// TwinCAT 3 PLC project Core
// Title: MTP
// Company: Zerlauth
// Author: Peter Zerlauth
// ProjectVersion: 0.0.0.0
// Description: Module Type Package MTP
// ProgramVersion: 3.1.4024.0
// libraries:
//   Tc2_Standard, * (Beckhoff Automation GmbH)
//   Tc2_System, * (Beckhoff Automation GmbH)
//   Tc2_Utilities, * (Beckhoff Automation GmbH)
// project tree:
//   Component/Event/ E_Event.TcDUT (not stored), E_Behaviour.TcDUT, FB_Event.TcPOU, I_Event.TcIO, ST_Event.TcDUT
//   Component/ E_Request.TcDUT (not stored), E_State.TcDUT, FB_Component.TcPOU, I_Component.TcIO
//   Component/Info/ FB_Info.TcPOU, I_Info.TcIO
//   Component/Observer/ FB_Observer.TcPOU, I_Observer.TcIO (not stored)
//   CyclicCall/ FB_Cycle.TcPOU, I_Cycle.TcIO
//   List/ FB_ListComponent.TcPOU (not stored), FB_ListObject.TcPOU, FB_ListString.TcPOU (not stored), I_ListComponent.TcIO (not stored), I_ListObject.TcIO, I_ListString.TcIO (not stored)
//   Logger/ FB_ListLogger.TcPOU, I_Logger.TcIO (not stored)
//   Object/ I_Object.TcIO (not stored)
//   Sequence/ FB_Sequence.TcPOU (not stored), I_Sequence.TcIO (not stored)
// (motion and I/O tree: see PLC project example)
// real-time tasks:
//   TASK plcTask1: cycle T#25000us, priority 20, ADS port 350

// ---- Component/Event/E_Behaviour.TcDUT
{attribute 'qualified_only'}
{attribute 'strict'}
{attribute 'to_string'}
TYPE E_Behaviour :
(
    Pause    := 100,
    Hold     := 200,    
	Complete := 300,	
    Stop  	 := 400,    
	Abort    := 500
 );	
END_TYPE

// ---- Component/Event/ST_Event.TcDUT
TYPE ST_Event :
STRUCT
	Source:			I_Component;
	EventType:		E_Event;
	Timestamp:   	ULINT;
	ID:				UDINT;
	Message:		STRING(255);
	Arguments:		STRING(255);
	Active:		BOOL;
END_STRUCT
END_TYPE

// ---- Component/E_State.TcDUT
{attribute 'qualified_only'}
{attribute 'strict'}
{attribute 'to_string'}
TYPE E_State :
(
	{attribute 'hide'}
	Undefined		:= 0,
	Idle			:= 1,
	
// Start
	Starting		:= 2,
	Execute			:= 3,
	
// Pause
	Pausing			:= 4,
	Paused			:= 5,
	Resuming		:= 6,
	
// Hold
	Holding			:= 7,
	Held			:= 8,
	Unholding		:= 9,
	
// Complete
	Completing		:= 10,
	Completed		:= 11,

// Stop
	Stopping		:= 12,
	Stopped			:= 13,

// Abort	
	Aborting		:= 14,
	Aborted			:= 15,

// Reset
	Resetting		:= 16

);
END_TYPE

// ---- Component/Event/I_Event.TcIO
INTERFACE I_Event EXTENDS I_Object

METHOD PUBLIC M_Debug : BOOL
VAR_INPUT
	Message:				STRING(255);
END_VAR
END_METHOD

METHOD PUBLIC M_Error : BOOL
VAR_INPUT
	Message:				STRING(255);
	ID:						UDINT;
	Behaviour:				E_Behaviour;
END_VAR
END_METHOD

METHOD PUBLIC M_Information : BOOL
VAR_INPUT
	Message:				STRING(255);
	ID:						UDINT;
END_VAR
END_METHOD

METHOD PUBLIC M_Warning : BOOL
VAR_INPUT
	Message:				STRING(255);
	ID:						UDINT;
END_VAR
END_METHOD

PROPERTY PUBLIC P_Logger : I_Logger
GET
END_GET
SET
END_SET
END_PROPERTY

END_INTERFACE

// ---- Component/Info/I_Info.TcIO
INTERFACE I_Info EXTENDS I_Object

PROPERTY PUBLIC P_Class : String(255)
GET
END_GET
END_PROPERTY

PROPERTY PUBLIC P_Comment : String(255)
GET
END_GET
END_PROPERTY

PROPERTY PUBLIC P_Instance : String(255)
GET
END_GET
END_PROPERTY

PROPERTY PUBLIC P_Timestamp : ULINT
GET
END_GET
END_PROPERTY

END_INTERFACE

// ---- Component/I_Component.TcIO
INTERFACE I_Component EXTENDS I_Object

METHOD PUBLIC M_OnNotify
VAR_INPUT
	eState:				E_State;
END_VAR
END_METHOD

METHOD PUBLIC M_Request : BOOL
VAR_INPUT
	eRequest:	E_Request;
END_VAR
END_METHOD

PROPERTY PUBLIC P_Event : I_Event
GET
END_GET
END_PROPERTY

PROPERTY PUBLIC P_Info : I_Info
GET
END_GET
END_PROPERTY

PROPERTY PUBLIC P_Observer : I_Observer
GET
END_GET
END_PROPERTY

PROPERTY PUBLIC P_State : E_State
GET
END_GET
END_PROPERTY

END_INTERFACE

// ---- CyclicCall/I_Cycle.TcIO
INTERFACE I_Cycle EXTENDS I_Object

END_INTERFACE

// ---- List/I_ListObject.TcIO
INTERFACE I_ListObject

METHOD PUBLIC M_Add : BOOL
VAR_INPUT
	Object: 	I_Object;
END_VAR
END_METHOD

METHOD PUBLIC M_Clear : BOOL
END_METHOD

METHOD PUBLIC M_Find : DINT
VAR_INPUT
	Object: 	I_Object;
END_VAR
END_METHOD

METHOD PUBLIC M_Index : I_Object
VAR_INPUT
	Index: 	DINT;
END_VAR
END_METHOD

METHOD PUBLIC M_Remove : BOOL
VAR_INPUT
	Object: 	I_Object;
END_VAR
END_METHOD

PROPERTY P_Length : DINT
GET
END_GET
END_PROPERTY

END_INTERFACE

// ---- Component/Event/FB_Event.TcPOU
FUNCTION_BLOCK FB_Event EXTENDS FB_ListString IMPLEMENTS I_Event
VAR_INPUT
	bIngoreHold:			BOOL:= TRUE;
	bIngorePause:			BOOL:= TRUE;
END_VAR
VAR_OUTPUT
END_VAR
VAR
	iParent:			I_Component;
	iLogger:			I_Logger;
	stEvent:			ST_Event;
END_VAR

SUPER^();

METHOD FB_init : BOOL
VAR_INPUT
	bInitRetains : BOOL; // if TRUE, the retain variables are initialized (warm start / cold start)
	bInCopyCode : BOOL;  // if TRUE, the instance afterwards gets moved into the copy code (online change)
	iParent:			I_Component;
END_VAR
THIS^.iParent:= iParent;
END_METHOD

METHOD INTERNAL M_Arguments : STRING(255)
VAR_INPUT
END_VAR
VAR
	nIndex:			INT;
END_VAR
WHILE nIndex < nLength DO
	M_Arguments:= Concat(Concat(M_Arguments, pList[nIndex]), '$N');
	nIndex:= nIndex + 1;
END_WHILE
END_METHOD

METHOD PUBLIC M_Debug : BOOL
VAR_INPUT
	Message:				STRING(255);
END_VAR
END_METHOD

METHOD PUBLIC M_Error : BOOL
VAR_INPUT
	Message:				STRING(255);
	ID:						UDINT;
	Behaviour:				E_Behaviour;
END_VAR
stEvent.Source:= iParent;
stEvent.EventType:= E_Event.Error;
stEvent.Timestamp:= F_GetSystemTime();
stEvent.ID:= ID;
stEvent.Message:= Message;
stEvent.Arguments:= M_Arguments();
stEvent.Active:= TRUE;

IF Behaviour >= E_Behaviour.Abort THEN
	iParent.M_Request(E_Request.Abort);
ELSIF Behaviour >= E_Behaviour.Stop THEN
	iParent.M_Request(E_Request.Stop);
ELSIF Behaviour >= E_Behaviour.Complete THEN	
	iParent.M_Request(E_Request.Complete);
ELSIF Behaviour >= E_Behaviour.Hold THEN
	iParent.M_Request(E_Request.Hold);
ELSIF Behaviour >= E_Behaviour.Pause THEN
	iParent.M_Request(E_Request.Pause);
END_IF

IF iLogger <> 0 THEN
	iLogger.M_Log(stEvent);
END_IF

M_Clear();
END_METHOD

METHOD PUBLIC M_Information : BOOL
VAR_INPUT
	Message:				STRING(255);
	ID:						UDINT;
END_VAR
END_METHOD

METHOD PUBLIC M_Warning : BOOL
VAR_INPUT
	Message:				STRING(255);
	ID:						UDINT;
END_VAR
END_METHOD

PROPERTY PUBLIC P_Logger : I_Logger
GET
P_Logger:= iLogger;
END_GET
SET
iLogger:= P_Logger;
END_SET
END_PROPERTY

END_FUNCTION_BLOCK

// ---- Component/FB_Component.TcPOU
{attribute 'reflection'} 
FUNCTION_BLOCK FB_Component EXTENDS FB_Cycle IMPLEMENTS I_Component
VAR_INPUT
	fbInfo:						FB_Info(sInstancePath);
	fbObserver:					FB_Observer;
	fbEvent:					FB_Event(THIS^);
END_VAR
VAR_OUTPUT
END_VAR
VAR
    {attribute 'hide'}
	{attribute 'instance-path'} 
    {attribute 'noinit'}
    sInstancePath:				STRING(255);	
	eRequest:					E_Request;
	eState:						E_State;
    {attribute 'hide'}
	eStatePrevious:				E_State;
END_VAR

METHOD PROTECTED M_Aborted : BOOL
VAR_INPUT
END_VAR
// State Aborted
M_Aborted:= True;
END_METHOD

METHOD PROTECTED M_Aborting : BOOL
VAR_INPUT
END_VAR
// State Aborting
M_Aborting:= True;
END_METHOD

METHOD PROTECTED M_Completed : BOOL
VAR_INPUT
END_VAR
// State Complete
M_Completed:= TRUE;
END_METHOD

METHOD PROTECTED M_Completing : BOOL
VAR_INPUT
END_VAR
// State Completing
M_Completing:= True;
END_METHOD

METHOD PUBLIC M_Cycle
VAR_INPUT
END_VAR
fbInfo();
fbObserver();
fbEvent();

// Handle Module Type Package states
CASE eState OF
	E_State.Undefined:
		IF M_Initialise() THEN
			eState:= E_State.Idle;					
		END_IF
		
	E_State.Resetting:
		CASE eRequest OF
			E_Request.Stop:
				eState:= E_State.Stopping;					
			E_Request.Abort:
				eState:= E_State.Aborting;						
		END_CASE	
		IF M_Resetting() THEN
			eState:= E_State.Idle;
		END_IF
		
	E_State.Idle:
		CASE eRequest OF
			E_Request.Start:
				eState:= E_State.Starting;
			E_Request.Stop:
				eState:= E_State.Stopping;					
			E_Request.Abort:
				eState:= E_State.Aborting;
			ELSE
				eRequest:= E_Request.Undefined;						
		END_CASE
		M_Idle();
		
	E_State.Starting:
		CASE eRequest OF
			E_Request.Stop:
				eState:= E_State.Stopping;					
			E_Request.Abort:
				eState:= E_State.Aborting;				
		END_CASE	
		IF M_Starting() THEN
			eState:= E_State.Execute;	
		END_IF		

	E_State.Execute:
		CASE eRequest OF
			E_Request.Pause:
				eState:= E_State.Pausing;		
			E_Request.Hold:
				eState:= E_State.Holding;		
			E_Request.Stop:
				eState:= E_State.Stopping;					
			E_Request.Abort:
				eState:= E_State.Aborting;
			ELSE
				eRequest:= E_Request.Undefined;						
		END_CASE
		IF M_Execute() THEN
			CASE eRequest OF
				E_Request.Complete:
					eState:= E_State.Completing;
			END_CASE	
		END_IF
		
	E_State.Stopping:
		CASE eRequest OF	
			E_Request.Abort:
				eState:= E_State.Aborting;			
		END_CASE	
		IF M_Stopping() THEN
			eState:= E_State.Stopped;
		END_IF

	E_State.Stopped:
		IF M_Stopped() THEN
			CASE eRequest OF
				E_Request.Reset:
					eState:= E_State.Resetting;
				ELSE
					eRequest:= E_Request.Undefined;	
			END_CASE		
		END_IF
		
	E_State.Aborting:
		IF M_Aborting() THEN
			eState:= E_State.Aborted;
		END_IF
		
	E_State.Aborted:
		IF M_Aborted() THEN
			CASE eRequest OF
				E_Request.Reset:
					eState:= E_State.Resetting;
				ELSE
					eRequest:= E_Request.Undefined;		
			END_CASE
		END_IF
		
	E_State.Pausing:
		CASE eRequest OF
			E_Request.Stop:
				eState:= E_State.Stopping;					
			E_Request.Abort:
				eState:= E_State.Aborting;					
		END_CASE	
		IF M_Pausing() THEN
			eState:= E_State.Paused;
		END_IF
	
	E_State.Paused:
		CASE eRequest OF
			E_Request.Stop:
				eState:= E_State.Stopping;					
			E_Request.Abort:
				eState:= E_State.Aborting;
			ELSE
				eRequest:= E_Request.Undefined;					
		END_CASE	
		IF M_Paused() THEN
			eState:= E_State.Resuming;			
		END_IF	
		
	E_State.Resuming:
		CASE eRequest OF
			E_Request.Stop:
				eState:= E_State.Stopping;					
			E_Request.Abort:
				eState:= E_State.Aborting;					
		END_CASE
		IF M_Resuming() THEN
			eState:= E_State.Execute;
		END_IF

	E_State.Holding:
		CASE eRequest OF
			E_Request.Stop:
				eState:= E_State.Stopping;					
			E_Request.Abort:
				eState:= E_State.Aborting;						
		END_CASE
		IF M_Holding() THEN
			eState:= E_State.Held;
		END_IF

	E_State.Held:
		CASE eRequest OF
			E_Request.Stop:
				eState:= E_State.Stopping;					
			E_Request.Abort:
				eState:= E_State.Aborting;
			ELSE
				eRequest:= E_Request.Undefined;					
		END_CASE
		IF M_Held() THEN
			eState:= E_State.Unholding;			
		END_IF	
		
	E_State.Unholding:
		CASE eRequest OF
			E_Request.Stop:
				eState:= E_State.Stopping;					
			E_Request.Abort:
				eState:= E_State.Aborting;							
		END_CASE
		IF M_Unholding() THEN
			eState:= E_State.Execute;
		END_IF
		
	E_State.Completing:
		CASE eRequest OF
			E_Request.Stop:
				eState:= E_State.Stopping;					
			E_Request.Abort:
				eState:= E_State.Aborting;				
		END_CASE
		IF M_Completing() THEN
			eState:= E_State.Completed;
		END_IF
		
	E_State.Completed:
		CASE eRequest OF
			E_Request.Stop:
				eState:= E_State.Stopping;					
			E_Request.Abort:
				eState:= E_State.Aborting;
			ELSE
				eRequest:= E_Request.Undefined;				
		END_CASE
		IF M_Completed() THEN
			CASE eRequest OF
				E_Request.Reset:	
					eState:= E_State.Resetting;
			END_CASE
		END_IF
		
	
END_CASE

CASE eState OF
	E_State.Aborted, E_State.Stopped, E_State.Completed:;
ELSE		
	this^.M_Running();
END_CASE

// Detect state changed
IF eStatePrevious <> eState THEN
	fbObserver.M_Notify(eState);
	eStatePrevious:= eState;
	M_OnStateChanged();
END_IF
END_METHOD

METHOD PROTECTED M_Execute : BOOL
VAR_INPUT
END_VAR
// State Execute
M_Execute:= TRUE;
END_METHOD

METHOD PROTECTED M_Held : BOOL
VAR_INPUT
END_VAR
// State Held
M_Held:= TRUE;
END_METHOD

METHOD PROTECTED M_Holding : BOOL
VAR_INPUT
END_VAR
// State Holding
M_Holding:= True;
END_METHOD

METHOD PROTECTED M_Idle : BOOL
VAR_INPUT
END_VAR
// State Idle
END_METHOD

METHOD PROTECTED M_Initialise : BOOL;
VAR_INPUT
END_VAR
// State Undefined
M_Initialise:= True;
END_METHOD

METHOD PUBLIC M_OnNotify
VAR_INPUT
	eState:				E_State;
END_VAR
CASE eState OF
	E_State.Undefined:;
	E_State.Idle:;
	E_State.Starting:
		M_Request(E_Request.Start);
	E_State.Execute:;
	E_State.Pausing:
		M_Request(E_Request.Pause);
	E_State.Paused:;
	E_State.Resuming:;
	E_State.Holding:
		M_Request(E_Request.Hold);
	E_State.Held:;
	E_State.Unholding:;
	E_State.Completing:
		M_Request(E_Request.Complete);
	E_State.Completed:;
	E_State.Stopping:
		M_Request(E_Request.Stop);
	E_State.Stopped:;
	E_State.Aborting:
		M_Request(E_Request.Abort);
	E_State.Aborted:;
	E_State.Resetting:
		M_Request(E_Request.Reset);
END_CASE
END_METHOD

METHOD PROTECTED M_OnStateChanged : BOOL
VAR_INPUT
END_VAR
END_METHOD

METHOD PROTECTED M_Paused : BOOL
VAR_INPUT
END_VAR
// State Held
M_Paused:= TRUE;
END_METHOD

METHOD PROTECTED M_Pausing : BOOL
VAR_INPUT
END_VAR
// State Holding
M_Pausing:= True;
END_METHOD

METHOD PUBLIC M_Request : BOOL
VAR_INPUT
	eRequest:	E_Request;
END_VAR
THIS^.eRequest:= eRequest;
CASE eRequest OF
	E_Request.Undefined:
		M_Request:= TRUE;
    E_Request.Start:
		M_Request:= eState = E_State.Execute;
    E_Request.Pause:
		IF 	fbEvent.bIngorePause THEN
			M_Request:= TRUE;
		ELSE
			M_Request:= eState = E_State.Paused;
		END_IF
    E_Request.Hold:
		IF 	fbEvent.bIngoreHold THEN
			M_Request:= TRUE;
		ELSE
			M_Request:= eState = E_State.Held;		
		END_IF
		
	E_Request.Complete:
		M_Request:= eState = E_State.Completed;	
    E_Request.Stop:
		M_Request:= eState = E_State.Stopped;	
	E_Request.Abort:
		M_Request:= eState = E_State.Aborted;	
	E_Request.Reset:
		M_Request:= eState = E_State.Idle;		

END_CASE
END_METHOD

METHOD PROTECTED M_Resetting : BOOL
VAR_INPUT
END_VAR
// State Resetting
M_Resetting:= True;
END_METHOD

METHOD PROTECTED M_Resuming : BOOL
VAR_INPUT
END_VAR
// State Holding
M_Resuming:= True;
END_METHOD

METHOD PROTECTED M_Running
VAR_INPUT
END_VAR
END_METHOD

METHOD PROTECTED M_Starting : BOOL
VAR_INPUT
END_VAR
// State Starting
M_Starting:= True;
END_METHOD

METHOD PROTECTED M_Stopped : BOOL
VAR_INPUT
END_VAR
// State Stopped
M_Stopped:= True;
END_METHOD

METHOD PROTECTED M_Stopping : BOOL
VAR_INPUT
END_VAR
// State Stopping
M_Stopping:= True;
END_METHOD

METHOD PROTECTED M_Unholding : BOOL
VAR_INPUT
END_VAR
// State Holding
M_Unholding:= True;
END_METHOD

PROPERTY PUBLIC P_Event : I_Event
GET
P_Event:= fbEvent;
END_GET
END_PROPERTY

PROPERTY PUBLIC P_Info : I_Info
GET
P_Info:= fbInfo;
END_GET
END_PROPERTY

PROPERTY PUBLIC P_Observer : I_Observer
GET
P_Observer:= fbObserver;
END_GET
END_PROPERTY

PROPERTY PUBLIC P_State : E_State
GET
P_State:= eState;
END_GET
END_PROPERTY

END_FUNCTION_BLOCK

// ---- CyclicCall/FB_Cycle.TcPOU
FUNCTION_BLOCK FB_Cycle IMPLEMENTS I_Cycle
VAR_INPUT
END_VAR
VAR_OUTPUT
END_VAR
VAR
END_VAR

METHOD PUBLIC M_Cycle
VAR_INPUT
END_VAR
END_METHOD

END_FUNCTION_BLOCK

// ---- Component/Info/FB_Info.TcPOU
FUNCTION_BLOCK PUBLIC FB_Info IMPLEMENTS I_Info
VAR_INPUT
END_VAR
VAR_OUTPUT
END_VAR
VAR
    sInstancePath:				REFERENCE TO STRING(255);
	fbReadSymInfo: 				PLC_ReadSymInfoByNameEx;
	nIndex:						DINT;
END_VAR
VAR_STAT
	nCycle: 					UDINT;
	nTimestamp: 				ULINT;
END_VAR

GETCURTASKINDEXEX(GETCURTASKINDEXEX => nIndex);
IF nCycle <> TwinCAT_SystemInfoVarList._TaskInfo[nIndex].CycleCount THEN
	nCycle:= TwinCAT_SystemInfoVarList._TaskInfo[nIndex].CycleCount;
	nTimestamp:= F_GetSystemTime();
END_IF

fbReadSymInfo(
	NETID:= , 
	PORT:= , 
	SYMNAME:= , 
	START:= , 
	TMOUT:= , 
	BUSY=> , 
	ERR=> , 
	ERRID=> , 
	SYMINFO=> , 
	OVTYPE=> , 
	OVCOMMENT=> );

METHOD FB_init : BOOL
VAR_INPUT
	bInitRetains : BOOL; // if TRUE, the retain variables are initialized (warm start / cold start)
	bInCopyCode : BOOL;  // if TRUE, the instance afterwards gets moved into the copy code (online change)
	sInstancePath:			REFERENCE TO STRING(255);
END_VAR
THIS^.sInstancePath REF= sInstancePath;
M_Initialize();
END_METHOD

METHOD PROTECTED M_Initialize
VAR_INPUT
END_VAR
VAR
    sName:				STRING(255);
    nPosition:			INT;
END_VAR
sName := CONCAT(TwinCAT_SystemInfoVarList._AppInfo.ProjectName, '.');

nPosition := FIND(sInstancePath, sName);
IF nPosition > 0 THEN
    fbReadSymInfo.SYMNAME:= DELETE(sInstancePath, nPosition-1 + LEN(sName), 1);
END_IF

nPosition := FIND(fbReadSymInfo.SYMNAME, sName);

IF nPosition > 0 THEN
    fbReadSymInfo.SYMNAME:= DELETE(fbReadSymInfo.SYMNAME, nPosition - 1 + LEN(sName), 1);
END_IF

fbReadSymInfo.PORT:= TwinCAT_SystemInfoVarList._AppInfo.AdsPort;
fbReadSymInfo.START:= TRUE;
END_METHOD

PROPERTY PUBLIC P_Class : String(255)
GET
P_Class:= fbReadSymInfo.SYMINFO.symDataType;
END_GET
END_PROPERTY

PROPERTY PUBLIC P_Comment : String(255)
GET
P_Comment:= fbReadSymInfo.SYMINFO.symComment;
END_GET
END_PROPERTY

PROPERTY PUBLIC P_Instance : String(255)
GET
P_Instance:= fbReadSymInfo.SYMNAME;
END_GET
END_PROPERTY

PROPERTY PUBLIC P_Timestamp : ULINT
GET
P_Timestamp:= nTimestamp;
END_GET
END_PROPERTY

END_FUNCTION_BLOCK

// ---- Component/Observer/FB_Observer.TcPOU
{attribute 'no_explicit_call'} 
FUNCTION_BLOCK PUBLIC FB_Observer IMPLEMENTS I_Observer
VAR
	pList: 			POINTER TO I_Component;
	nLength:		DINT;
	aList:			POINTER TO POINTER TO ARRAY [0..100] OF I_Component:=ADR(pList);
END_VAR

METHOD FB_exit : BOOL
VAR_INPUT
	bInCopyCode : BOOL; // if TRUE, the exit method is called for exiting an instance that is copied afterwards (online change).
END_VAR
M_Clear();
END_METHOD

METHOD M_Attach : BOOL
VAR_INPUT
	Object: 	I_Component;
END_VAR
VAR
	pOldList: 	POINTER TO I_Component;
END_VAR
IF Object <> 0 THEN
	// First Item
	IF pList = 0 THEN
		nLength:= nLength + 1;
		pList:= __NEW(POINTER TO I_Component,DINT_TO_UDINT(nLength));
	ELSE
		// Item already in List
		IF M_Find(Object) = -1 THEN
			// backup 
			pOldList:= pList;
			// new Length
			nLength:= nLength + 1;
			// new pointer
			pList:= __NEW(POINTER TO I_Component,DINT_TO_UDINT(nLength));
			// restore
			Memcpy(pList,pOldList, SIZEOF(POINTER TO I_Component)*DINT_TO_UDINT(nLength -1));
			// delete old
			__DELETE(pOldList);
		ELSE
			M_Attach:= FALSE;	
			RETURN;
		END_IF
	END_IF
	IF pList = 0 THEN
		RETURN;
	END_IF
	// add new Object
	pList[nLength-1]:= Object;
	M_Attach:= TRUE;
ELSE
	M_Attach:= FALSE;	
END_IF
END_METHOD

METHOD M_Clear
IF pList <> 0 THEN
	nLength:= 0;
	__DELETE(pList);
END_IF
END_METHOD

METHOD M_Detach : BOOL
VAR_INPUT
	Object: 	I_Component;
END_VAR
VAR
	pOldList:			POINTER TO I_Component;
	nPosition: 			DINT;
END_VAR
IF Object <> 0 THEN
	// First Item
	IF nLength >= 0 THEN
		// Item already in List
		nPosition:= M_Find(Object);
		IF nPosition <> -1 THEN
			// backup 
			pOldList:= pList;
			// new Length
			nLength:= nLength -1;
			// new pointer
			pList:= __NEW(POINTER TO I_Component,DINT_TO_UDINT(nLength));
			// restore lower part
			Memcpy(pList,pOldList, SIZEOF(POINTER TO I_Component) * DINT_TO_UDINT(nPosition));
			//pList[nPosition]:= iObject;
			Memcpy(pList + (SIZEOF(POINTER TO I_Component)*nPosition),pOldList + (SIZEOF(POINTER TO I_Component)*(nPosition + 1)), SIZEOF(POINTER TO I_Component) * DINT_TO_UDINT(nLength - nPosition));
			// delete old
			__DELETE(pOldList);
		ELSE
			M_Detach:= FALSE;	
			RETURN;
		END_IF
	ELSE
		M_Detach:= FALSE;	
		RETURN;
	END_IF
	M_Detach:= TRUE;
ELSE
	M_Detach:= FALSE;	
END_IF
END_METHOD

METHOD M_Find : DINT
VAR_INPUT
	Object: 	I_Component;
END_VAR
VAR
	nIndex: 	UINT;
END_VAR
// Object already in List
M_Find := -1;
WHILE nIndex < nLength DO
    IF (pList[nIndex] = Object) THEN
        M_Find := nIndex;
        RETURN;
    END_IF
	nIndex := nIndex + 1;
END_WHILE
END_METHOD

METHOD M_Index : I_Component
VAR_INPUT
	Index: 	DINT;
END_VAR
IF Index <= nLength THEN
	M_Index:= pList[Index];
END_IF
END_METHOD

METHOD M_Notify : BOOL
VAR_INPUT
	eRequest:		E_Request;
END_VAR

VAR
	nIndex: 	INT;
END_VAR
WHILE nIndex < nLength DO
	pList[nIndex].M_OnNotify(eRequest);
	nIndex:= nIndex + 1; 
END_WHILE
END_METHOD

PROPERTY P_Length : DINT
GET
P_Length:= nLength;
END_GET
END_PROPERTY

END_FUNCTION_BLOCK

// ---- List/FB_ListObject.TcPOU
{attribute 'no_explicit_call'} 
FUNCTION_BLOCK FB_ListObject IMPLEMENTS I_ListObject
VAR
	nLength:		DINT;
	pList: 			POINTER TO I_Object;
	{attribute 'conditionalshow'}
	aList:			POINTER TO POINTER TO ARRAY [0..100] OF I_Object:=ADR(pList);
END_VAR

METHOD FB_exit : BOOL
VAR_INPUT
	bInCopyCode : BOOL; // if TRUE, the exit method is called for exiting an instance that is copied afterwards (online change).
END_VAR
M_Clear();
END_METHOD

METHOD PUBLIC M_Add : BOOL
VAR_INPUT
	Object: 	I_Object;
END_VAR
VAR
	pOldList: 	POINTER TO I_Object;
END_VAR
IF Object <> 0 THEN
	// First Item
	IF pList = 0 THEN
		nLength:= nLength + 1;
		pList:= __NEW(POINTER TO I_Object,DINT_TO_UDINT(nLength));
	ELSE
		// Item already in List
		IF M_Find(Object) = -1 THEN
			// backup 
			pOldList:= pList;
			// new Length
			nLength:= nLength + 1;
			// new pointer
			pList:= __NEW(POINTER TO I_Object,DINT_TO_UDINT(nLength));
			// restore
			Memcpy(pList,pOldList, SIZEOF(POINTER TO I_Object)*DINT_TO_UDINT(nLength -1));
			// delete old
			__DELETE(pOldList);
		ELSE
			M_Add:= FALSE;	
			RETURN;
		END_IF
	END_IF
	IF pList = 0 THEN
		RETURN;
	END_IF
	// add new Object
	pList[nLength-1]:= Object;
	M_Add:= TRUE;
ELSE
	M_Add:= FALSE;	
END_IF
END_METHOD

METHOD PUBLIC M_Clear : bool
IF pList <> 0 THEN
	nLength:= 0;
	__DELETE(pList);
END_IF
M_Clear:= True;
END_METHOD

METHOD PUBLIC M_Find : DINT
VAR_INPUT
	Object: 	I_Object;
END_VAR
VAR
	nIndex: 	UINT;
END_VAR
// Object already in List
M_Find := -1;
WHILE nIndex < nLength DO
    IF (pList[nIndex] = Object) THEN
        M_Find := nIndex;
        RETURN;
    END_IF
	nIndex := nIndex + 1;
END_WHILE
END_METHOD

METHOD PUBLIC M_Index : I_Object
VAR_INPUT
	Index: 	DINT;
END_VAR
IF Index <= nLength THEN
	M_Index:= pList[Index];
END_IF
END_METHOD

METHOD PUBLIC M_Remove : BOOL
VAR_INPUT
	Object: 	I_Object;
END_VAR
VAR
	pOldList:			POINTER TO I_Object;
	nPosition: 			DINT;
END_VAR
IF Object <> 0 THEN
	// First Item
	IF nLength >= 0 THEN
		// Item already in List
		nPosition:= M_Find(Object);
		IF nPosition <> -1 THEN
			// backup 
			pOldList:= pList;
			// new Length
			nLength:= nLength -1;
			// new pointer
			pList:= __NEW(POINTER TO I_Object,DINT_TO_UDINT(nLength));
			// restore lower part
			Memcpy(pList,pOldList, SIZEOF(POINTER TO I_Object) * DINT_TO_UDINT(nPosition));
			//pList[nPosition]:= iObject;
			Memcpy(pList + (SIZEOF(POINTER TO I_Object)*nPosition),pOldList + (SIZEOF(POINTER TO I_Object)*(nPosition + 1)), SIZEOF(POINTER TO I_Object) * DINT_TO_UDINT(nLength - nPosition));
			// delete old
			__DELETE(pOldList);
		ELSE
			M_Remove:= FALSE;	
			RETURN;
		END_IF
	ELSE
		M_Remove:= FALSE;	
		RETURN;
	END_IF
	M_Remove:= TRUE;
ELSE
	M_Remove:= FALSE;	
END_IF
END_METHOD

PROPERTY PUBLIC P_Length : DINT
GET
P_Length:= nLength;
END_GET
END_PROPERTY

END_FUNCTION_BLOCK

// ---- Logger/FB_ListLogger.TcPOU
{attribute 'no_explicit_call'} 
FUNCTION_BLOCK FB_ListLogger IMPLEMENTS I_Logger
VAR
	pList: 			POINTER TO I_Logger;
	nLength:		DINT;
	{attribute 'conditionalshow'}
	aList:			POINTER TO POINTER TO ARRAY [0..100] OF I_Logger:=ADR(pList);
END_VAR

METHOD FB_exit : BOOL
VAR_INPUT
	bInCopyCode : BOOL; // if TRUE, the exit method is called for exiting an instance that is copied afterwards (online change).
END_VAR
M_Clear();
END_METHOD

METHOD M_Add : BOOL
VAR_INPUT
	Object: 	I_Logger;
END_VAR
VAR
	pOldList: 	POINTER TO I_Logger;
END_VAR
IF Object <> 0 THEN
	// First Item
	IF pList = 0 THEN
		nLength:= nLength + 1;
		pList:= __NEW(POINTER TO I_Logger,DINT_TO_UDINT(nLength));
	ELSE
		// Item already in List
		IF M_Find(Object) = -1 THEN
			// backup 
			pOldList:= pList;
			// new Length
			nLength:= nLength + 1;
			// new pointer
			pList:= __NEW(POINTER TO I_Object,DINT_TO_UDINT(nLength));
			// restore
			Memcpy(pList,pOldList, SIZEOF(POINTER TO I_Logger)*DINT_TO_UDINT(nLength -1));
			// delete old
			__DELETE(pOldList);
		ELSE
			M_Add:= FALSE;	
			RETURN;
		END_IF
	END_IF
	IF pList = 0 THEN
		RETURN;
	END_IF
	// add new Object
	pList[nLength-1]:= Object;
	M_Add:= TRUE;
ELSE
	M_Add:= FALSE;	
END_IF
END_METHOD

METHOD M_Clear : bool
IF pList <> 0 THEN
	nLength:= 0;
	__DELETE(pList);
END_IF
M_Clear:= True;
END_METHOD

METHOD M_Find : DINT
VAR_INPUT
	Object: 	I_Logger;
END_VAR
VAR
	nIndex: 	UINT;
END_VAR
// Object already in List
M_Find := -1;
WHILE nIndex < nLength DO
    IF (pList[nIndex] = Object) THEN
        M_Find := nIndex;
        RETURN;
    END_IF
	nIndex := nIndex + 1;
END_WHILE
END_METHOD

METHOD M_Index : I_Logger
VAR_INPUT
	Index: 	DINT;
END_VAR
IF Index <= nLength THEN
	M_Index:= pList[Index];
END_IF
END_METHOD

METHOD PUBLIC M_Log
VAR_INPUT
	stEvent:		ST_Event;
END_VAR

VAR
	nIndex: INT;
END_VAR
WHILE nIndex < nLength DO
	M_Index(nIndex).M_Log(stEvent);
	nIndex:= nIndex +1;
END_WHILE
END_METHOD

METHOD M_Remove : BOOL
VAR_INPUT
	Object: 	I_Logger;
END_VAR
VAR
	pOldList:			POINTER TO I_Logger;
	nPosition: 			DINT;
END_VAR
IF Object <> 0 THEN
	// First Item
	IF nLength >= 0 THEN
		// Item already in List
		nPosition:= M_Find(Object);
		IF nPosition <> -1 THEN
			// backup 
			pOldList:= pList;
			// new Length
			nLength:= nLength -1;
			// new pointer
			pList:= __NEW(POINTER TO I_Logger,DINT_TO_UDINT(nLength));
			// restore lower part
			Memcpy(pList,pOldList, SIZEOF(POINTER TO I_Logger) * DINT_TO_UDINT(nPosition));
			//pList[nPosition]:= iObject;
			Memcpy(pList + (SIZEOF(POINTER TO I_Logger)*nPosition),pOldList + (SIZEOF(POINTER TO I_Logger)*(nPosition + 1)), SIZEOF(POINTER TO I_Logger) * DINT_TO_UDINT(nLength - nPosition));
			// delete old
			__DELETE(pOldList);
		ELSE
			M_Remove:= FALSE;	
			RETURN;
		END_IF
	ELSE
		M_Remove:= FALSE;	
		RETURN;
	END_IF
	M_Remove:= TRUE;
ELSE
	M_Remove:= FALSE;	
END_IF
END_METHOD

PROPERTY P_Length : DINT
GET
P_Length:= nLength;
END_GET
END_PROPERTY

END_FUNCTION_BLOCK
